FUNCTION_BLOCK FB_Mechinit EXTENDS CycleHandleFB
VAR_INPUT
	Ctrl_ref:			REFERENCE TO Ctrl_Typ;
END_VAR
VAR_OUTPUT
END_VAR
VAR
	MethInitDone:		BOOL;
END_VAR

VAR CONSTANT
// States are global
		
	MECHINIT_INIT:							INT:=0;
	MECHINIT_SWITCH_ON:						INT:=10;
	MECHINIT_RUN_MASTER:					INT:=20;
	MECHINIT_GEAR_IN:						INT:=30;
	MECHINIT_DONE:							INT:=100;
END_VAR

	IF NOT MethInitDone THEN
		MethInitDone	:= Meth_Init();
	END_IF
	
	IF  THIS^.CMD.Pause = FALSE THEN
		
		//-----------------------------
		//State Machine
		//-----------------------------
		CASE THIS^.StepNo OF
			MECHINIT_INIT:
				IF THIS^.StepOneShotTrig THEN
					THIS^.Monitoring.StepMessage	:= 'Init: Start.';
					THIS^.Delay(IN:=FALSE);
				ELSIF Meth_Enable(TRUE) THEN
					THIS^.StepNo	:= 	MECHINIT_SWITCH_ON;
				END_IF
			
			MECHINIT_SWITCH_ON:
				IF THIS^.StepOneShotTrig THEN
					THIS^.Monitoring.StepMessage	:= 'Switch motor on.';
					THIS^.Delay(IN:=FALSE);
					Meth_SwitchOn(FALSE);
				ELSIF Meth_SwitchOn(TRUE) THEN
					THIS^.StepNo	:= 	MECHINIT_RUN_MASTER;
				END_IF	
				
			MECHINIT_RUN_MASTER:
				IF THIS^.StepOneShotTrig THEN
					THIS^.Monitoring.StepMessage	:= 'Start master';
					THIS^.Delay(IN:=FALSE);
					Meth_StartVmaster(FALSE);
				ELSIF Meth_StartVmaster(TRUE) THEN
					THIS^.StepNo	:= 	MECHINIT_GEAR_IN;
				END_IF				
				

			MECHINIT_GEAR_IN:
				IF THIS^.StepOneShotTrig THEN
					THIS^.Monitoring.StepMessage	:= 'Gear In';
					THIS^.Delay(IN:=FALSE);
					Meth_GearIn(FALSE);
				ELSIF Meth_GearIn(TRUE) THEN
					THIS^.StepNo	:= 	MECHINIT_DONE;
				END_IF	
				
				
			MECHINIT_DONE:
				IF THIS^.StepOneShotTrig THEN
					THIS^.Monitoring.StepMessage	:= 'mechinit cycle Done';
				ELSIF Meth_Done(TRUE) THEN
					THIS^.StepNo	:= 	MECHINIT_INIT;
				END_IF					
				
		END_CASE
	
	ELSE
		THIS^.Monitoring.StepMessage:= 'Pause';
		
		IF THIS^.Status.Fault = TRUE THEN
		//IF Meth_EmStop(TRUE) THEN
				THIS^.CMD.ResetCycle	:= TRUE;		// Reset the all state machine to start point
		//END_IF
			
		END_IF
		
	END_IF
	
	THIS^.Delay();
	THIS^.CH_Logic();
	
	// Reset Meth_EmStop when at Init State
	IF THIS^.Pause = FALSE THEN
		//Meth_EmStop(FALSE);
	END_IF

METHOD PRIVATE Meth_Done : BOOL
VAR_INPUT
	Execute: 	BOOL;
END_VAR


	//THIS^.Monitoring.StepMessage			:= 'Press 1 engage';
	//THIS^.Monitoring.Error_Text				:= 'Press 1 engage Fail';
	//THIS^.CMD.Deacivate_Sequence_Time_Out	:= TRUE;	// Disable time out to the all sequence
	//THIS^.CMD.DeactivateStepTimeOut			:= TRUE;	// Disable time out to the actual step
	//THIS^.Parameter.TimeOut					:= T#5S;

	THIS^.Status.Done		:= TRUE;
	THIS^.Status.Running	:= FALSE;									
	Meth_Done	:= TRUE;
END_METHOD

METHOD PRIVATE Meth_Enable : BOOL
VAR_INPUT
	Execute: 	BOOL;
END_VAR


IF THIS^.CMD.Start THEN
	
	THIS^.Monitoring.StepMessage			:= 'Start';
	THIS^.Monitoring.Error_Text				:= 'Start Fail';
	THIS^.CMD.Deacivate_Sequence_Time_Out	:= TRUE;	// Disable time out to the all sequence
	THIS^.CMD.DeactivateStepTimeOut			:= TRUE;	// Disable time out to the actual step
	THIS^.Parameter.TimeOut					:= T#0.5S;

	THIS^.CMD.Start			:= FALSE;
	THIS^.Status.Done		:= FALSE;
	THIS^.Status.Running	:= TRUE;
	
	// Reset Commands and Statuses												
	
	Meth_Enable	:= TRUE;
END_IF
END_METHOD

METHOD Meth_GearIn : BOOL
VAR_INPUT
	Execute: 	BOOL;
END_VAR
VAR_INST	
	ExecuteTrig: 	Trigger;	
END_VAR
IF ExecuteTrig.EDGEPOS(Execute) THEN
	Meth_GearIn	:= FALSE;
	THIS^.SubStepNo:= 	1;	
END_IF

IF ExecuteTrig.EDGENEG(Execute) THEN
	Meth_GearIn	:=	FALSE;
END_IF

CASE THIS^.SubStepNo OF
	   
	1:
		THIS^.Monitoring.StepMessage:= 'Set GearInMultiMaster command';
		
		gWebAxes.UW_1.Crtl.MultiAxis.Input.Parameter.GearInMultiMaster.GearRatio1:=	0;

		
		gWebAxes.UW_1.Crtl.MultiAxis.Input.Parameter.GearInMultiMaster.Acceleration:= 	1000000;
		gWebAxes.UW_1.Crtl.MultiAxis.Input.Parameter.GearInMultiMaster.Deceleration:= 	1000000;
		gWebAxes.UW_1.Crtl.MultiAxis.Input.Parameter.GearInMultiMaster.Jerk:=			0;
		gWebAxes.UW_1.Crtl.MultiAxis.Input.Parameter.GearInMultiMaster.Options.AdvancedSlaveDynamics:= 	FALSE;
		
		gWebAxes.UW_1.Crtl.MultiAxis.Input.Command.GearInMultiMaster.StartSlave:=		TRUE;
				
								
		THIS^.SubStepNo	:= 2;		
			
	2:	
		THIS^.Monitoring.StepMessage:= 	'Wait for GearInMultiMaster done UW1' ;
							
		IF (gWebAxes.UW_1.Crtl.MultiAxis.Input.Command.GearInMultiMaster.StartSlave = FALSE) 
			AND (gWebAxes.UW_1.Crtl.MultiAxis.Output.Status.GearInMultiMaster.InGear = TRUE) THEN
			THIS^.SubStepNo:=	3;
		ELSIF 	gWebAxes.UW_1.Crtl.MultiAxis.Output.Status.GearInMultiMaster.InGear = TRUE THEN
			THIS^.SubStepNo:=	3;
		END_IF		


	3:
		THIS^.Monitoring.StepMessage:= 'Set GearInMultiMaster UW2 command';
		
		gWebAxes.UW_2.Crtl.MultiAxis.Input.Parameter.GearInMultiMaster.GearRatio1:=	0;

		
		gWebAxes.UW_2.Crtl.MultiAxis.Input.Parameter.GearInMultiMaster.Acceleration:= 	1000000;
		gWebAxes.UW_2.Crtl.MultiAxis.Input.Parameter.GearInMultiMaster.Deceleration:= 	1000000;
		gWebAxes.UW_2.Crtl.MultiAxis.Input.Parameter.GearInMultiMaster.Jerk:=			0;
		gWebAxes.UW_2.Crtl.MultiAxis.Input.Parameter.GearInMultiMaster.Options.AdvancedSlaveDynamics:= 	FALSE;
		
		gWebAxes.UW_2.Crtl.MultiAxis.Input.Command.GearInMultiMaster.StartSlave:=		TRUE;
				
								
		THIS^.SubStepNo	:= 4;		
			
	4:	
		THIS^.Monitoring.StepMessage:= 	'Wait for GearInMultiMaster done' ;
							
		IF (gWebAxes.UW_2.Crtl.MultiAxis.Input.Command.GearInMultiMaster.StartSlave = FALSE) 
			AND (gWebAxes.UW_2.Crtl.MultiAxis.Output.Status.GearInMultiMaster.InGear = TRUE) THEN
			THIS^.SubStepNo:=	0;
			Meth_GearIn:= 	TRUE;
		ELSIF gWebAxes.UW_2.Crtl.MultiAxis.Output.Status.GearInMultiMaster.InGear = TRUE THEN	
			THIS^.SubStepNo:=	0;
			Meth_GearIn:= 	TRUE;
		END_IF	

							
END_CASE
END_METHOD

METHOD Meth_Init :BOOL
VAR_INPUT
END_VAR
//resets


Meth_Init:=TRUE;
END_METHOD

METHOD Meth_StartVmaster : BOOL
VAR_INPUT
	Execute: 	BOOL;
END_VAR
VAR_INST	
	ExecuteTrig: 	Trigger;	
END_VAR

IF ExecuteTrig.EDGEPOS(Execute) THEN
	Meth_StartVmaster	:= FALSE;
	THIS^.SubStepNo:= 	1;	
END_IF

IF ExecuteTrig.EDGENEG(Execute) THEN
	Meth_StartVmaster	:=	FALSE;
END_IF


CASE THIS^.SubStepNo OF
	   
	1:
		THIS^.Monitoring.StepMessage	:= 'Set RunVel command to Master Tension';
		
			gWebAxes.UwVmaster.Crtl.Basic_axis.Input.Parameter.Acceleration	:= 100000; 
			gWebAxes.UwVmaster.Crtl.Basic_axis.Input.Parameter.Deceleration	:= 100000; 
			gWebAxes.UwVmaster.Crtl.Basic_axis.Input.Parameter.Velocity		:= 360000;//100000 
			gWebAxes.UwVmaster.Crtl.Basic_axis.Input.Parameter.Direction		:= MC_Positive_Direction; 		
				
			gWebAxes.UwVmaster.Crtl.Basic_axis.Input.Command.MoveVelocity		:= TRUE;
			THIS^.SubStepNo:= 	2;	

	2:	
		THIS^.Monitoring.StepMessage	:= 'Wait @ velocity from Master';
		IF (gWebAxes.UwVmaster.Crtl.Basic_axis.Output.Status.AxisStatus.ContinuousMotion = TRUE) THEN	
			Meth_StartVmaster:=TRUE;
			THIS^.SubStepNo:= 	0;				
		END_IF
								
END_CASE
END_METHOD

METHOD Meth_SwitchOn : BOOL
VAR_INPUT
	Execute: 	BOOL;
END_VAR
VAR_INST
	ExecuteTrig: 	Trigger;
END_VAR


IF ExecuteTrig.EDGEPOS(Execute) THEN
	Meth_SwitchOn:=	FALSE;
	THIS^.SubStepNo:= 	1;	
END_IF

IF ExecuteTrig.EDGENEG(Execute) THEN
	Meth_SwitchOn:=	FALSE;
END_IF

CASE THIS^.SubStepNo OF
	(* Power ON*)
	1:
		THIS^.Monitoring.StepMessage	:= 'Power On';								
		gWebAxes.UW_1.Crtl.Basic_axis.Input.Command.Power		:= TRUE;
		gWebAxes.UW_2.Crtl.Basic_axis.Input.Command.Power		:= TRUE;	
		gWebAxes.UwVmaster.Crtl.Basic_axis.Input.Command.Power	:= TRUE;
		
		THIS^.SubStepNo:= 2;		
	
	2:	
		THIS^.Monitoring.StepMessage:= 'Wait for standstill UW 1';
									
		IF gWebAxes.UW_1.Crtl.Basic_axis.Output.Status.AxisStatus.StandStill
		OR gWebAxes.UW_1.Crtl.Basic_axis.Output.Status.AxisStatus.SynchronizedMotion THEN
			THIS^.SubStepNo	:= 3 ;
		END_IF
		
	3:	
		THIS^.Monitoring.StepMessage:= 'Wait for standstill UW 2';
									
		IF gWebAxes.UW_2.Crtl.Basic_axis.Output.Status.AxisStatus.StandStill
		OR  gWebAxes.UW_2.Crtl.Basic_axis.Output.Status.AxisStatus.SynchronizedMotion THEN
			THIS^.SubStepNo	:= 4 ;
		END_IF		
		
	4:	
		THIS^.Monitoring.StepMessage:= 'Wait for standstill from master';
									
		IF gWebAxes.UwVmaster.Crtl.Basic_axis.Output.Status.AxisStatus.StandStill
		OR  gWebAxes.UwVmaster.Crtl.Basic_axis.Output.Status.AxisStatus.ContinuousMotion THEN
			THIS^.SubStepNo	:= 10 ;
			Meth_SwitchOn	:= TRUE;
		END_IF
							
END_CASE
END_METHOD

END_FUNCTION_BLOCK

(* stored: Version 1.1.0.1, ProductVersion 3.1.4024.3
   POU FB_Mechinit: Id {45179798-8c3f-447d-8c4a-8963e3104817}, SpecialFunc None
   Method Meth_Done: Id {a7b5a54f-c321-4b1c-b7ae-c1c5d5459d19}
   Method Meth_Enable: Id {d02e2caa-073e-4212-8302-a5caacdaf860}
   Method Meth_GearIn: Id {03ab5f7c-9a27-4239-a28a-13b70cfd59cc}
   Method Meth_Init: Id {5392863f-8e40-46d6-90d2-4f5b46866e43}
   Method Meth_StartVmaster: Id {f812e205-dcf6-40f1-b43f-2a81c2f34576}
   Method Meth_SwitchOn: Id {a122ecf0-6b0c-4f90-92e6-2b6c9d30b5f1} *)
